PROGRAM MAIN
VAR
END_VAR

PRG_PythonServerConnect();

END_PROGRAM

(* stored: Version 1.1.0.1, ProductVersion 3.1.4024.11
   POU MAIN: Id {0aa57708-3cf4-4eb6-950e-a14cb0a5b886}, SpecialFunc None *)
